// Block: Straightener_PERS

DATA_BLOCK Straightener_PERS
VERSION : 0.1
   NON_RETAIN
   VAR
      PersistentValues : Struct
         Data : Struct
            Feed : PositioningMachine_DataPers;
         END_STRUCT;
         Feed : PositioningMachine_Par;
      END_STRUCT;
   END_VAR

BEGIN
   // No initialization required
END_DATA_BLOCK
